FUNCTION_BLOCK PUBLIC FB_CylinderDriver EXTENDS FB_ComponentBase IMPLEMENTS ITF_Cylinder, ITFComponent
VAR_INPUT
	bSafetyOk				: BOOL; // Freigabe von Sicherheit
	
	bEnableHp				: BOOL;	// Freigabe Grundposition
	bEnableWp				: BOOL;	// Freigabe Arbeitsposition
END_VAR
VAR_OUTPUT
	// Zylinder ist in Grundstellung (verzögert)
	bIsInHp	: BOOL;
	// Zylinder ist in Arbeitsstellung (verzögert)
	bIsInWp	: BOOL;
	// Zylinder Ist-Position
	eActPos	: E_CylinderPosition;
END_VAR
VAR
	/// IO reference
	stIn 	: REFERENCE TO ST_CylinderDriverIn;
	stOut 	: REFERENCE TO ST_CylinderDriverOut;
	
	bWpSensor				: BOOL := TRUE;
	bHpSensor				: BOOL := TRUE;
	
	// private var's
	eReqPos					: E_CylinderPosition;	// Zylinder Soll-Position
	fPositionValidationTime	: TIME := T#300MS; 		// Verweilzeit bis die jeweilige Endlage bestätigt wird.
	tImpulseTime 			: TIME := T#0S; 		// Ansteuerzeit für Impulsventile (0 deaktiviert die Impulssteuerung)
	fSupervisionTime		: TIME := T#5S; 		// Verweilzeit nach Ventilansteuerung, bis die Zylinderendlage geprüft wird (0 deaktiviert die Überwachung)
	tonValveChange			: TON;					// Zeit seit Veränderung der Ventilstellung
	tonIsInHp				: TON;					// Verzögerung in Grundstellung
	tonIsInWp				: TON;					// Verzögerung in Arbeitsstellung
END_VAR

///
/// Cylinder driver FB
/// TP/www.rmth.at/06.2015
///

PROPERTY PUBLIC ActualPosition : E_CylinderPosition
GET
ActualPosition := eActPos;
END_GET
END_PROPERTY

PROPERTY PUBLIC EnableHp : BOOL
GET
EnableHp := bEnableHp;
END_GET
SET
bEnableHp := EnableHp;
END_SET
END_PROPERTY

PROPERTY PUBLIC EnableHpSensor : BOOL
GET
EnableHpSensor := bHpSensor;
END_GET
SET
bHpSensor := EnableHpSensor;
END_SET
END_PROPERTY

PROPERTY PUBLIC EnableWp : BOOL
GET
EnableWp := bEnableWp;
END_GET
SET
bEnableWp := EnableWp;
END_SET
END_PROPERTY

PROPERTY PUBLIC EnableWpSensor : BOOL
GET
EnableWpSensor := bWpSensor;
END_GET
SET
bWpSensor := EnableWpSensor;
END_SET
END_PROPERTY

METHOD FB_init : BOOL
VAR_INPUT
	bInitRetains : BOOL; // if TRUE, the retain variables are initialized (warm start / cold start)
	bInCopyCode : BOOL;  // if TRUE, the instance afterwards gets moved into the copy code (online change)
END_VAR
eTyp := E_ComponentType.eComponentType_Cylinder;
END_METHOD

// Ansteuerzeit für Impulsventile (0 deaktiviert die Impulssteuerung)
PROPERTY PUBLIC ImpulseTime : TIME
GET
// Ansteuerzeit für Impulsventile (0 deaktiviert die Impulssteuerung)
ImpulseTime := tImpulseTime;
END_GET
SET
// Ansteuerzeit für Impulsventile (0 deaktiviert die Impulssteuerung)
tImpulseTime := ImpulseTime;
END_SET
END_PROPERTY

/// Verweilzeit bis die jeweilige Endlage bestätigt wird.
PROPERTY PUBLIC PositionValidationTime : TIME
GET
/// Verweilzeit bis die jeweilige Endlage bestätigt wird.
PositionValidationTime := fPositionValidationTime;
END_GET
SET
/// Verweilzeit bis die jeweilige Endlage bestätigt wird.
fPositionValidationTime := PositionValidationTime;
END_SET
END_PROPERTY

PROPERTY PUBLIC RequestPosition : E_CylinderPosition
GET
RequestPosition := eReqPos;
END_GET
END_PROPERTY

METHOD Reset
VAR_INPUT
END_VAR
// base logic run
SUPER^.Reset();

//ToHP();
tonValveChange(IN := FALSE);
tonIsInHp(IN := FALSE);
tonIsInWp(IN := FALSE);

eState := E_ComponentState.eComponentState_ready;
END_METHOD

METHOD PUBLIC ResetValves
VAR_INPUT
END_VAR
IF NOT __ISVALIDREF(stOut) THEN
	sLastError := 'IO reference not set';
	eState := E_ComponentState.eComponentState_error;
	RETURN;
END_IF

// chk
IF NOT bSafetyOk THEN
	sClearText := 'Warte auf Sicherheit Ok';
	RETURN;
END_IF

eReqPos := eCylinderPosition_unknown;
stOut.bValveCylinderHp := FALSE;
stOut.bValveCylinderWp := FALSE;
tonValveChange(IN := FALSE);
END_METHOD

/// Run component logic
{attribute 'object_name' := 'Run'}
METHOD Run : E_ComponentState
// base logic run
Run := SUPER^.Run();

// chk
IF NOT (__ISVALIDREF(stIn) AND __ISVALIDREF(stOut)) THEN
	sLastError := 'IO reference not set';
	eState := E_ComponentState.eComponentState_error;
	RETURN;
END_IF



// definiere aktuelle Zylinderposition
IF (stIn.bCylinderSensorHp OR (NOT bHpSensor AND stOut.bValveCylinderHp)) AND NOT stIn.bCylinderSensorWp THEN
	eActPos := eCylinderPosition_hp;
ELSIF NOT stIn.bCylinderSensorHp AND (stIn.bCylinderSensorWp OR (NOT bWpSensor AND stOut.bValveCylinderWp)) THEN
	eActPos := eCylinderPosition_wp;
ELSE
	eActPos := eCylinderPosition_unknown;
END_IF

tonIsInHp(IN := (eActPos = eCylinderPosition_hp), PT := fPositionValidationTime);
bIsInHp := tonIsInHp.Q;

tonIsInWp(IN := (eActPos = eCylinderPosition_wp), PT := fPositionValidationTime);
bIsInWp := tonIsInWp.Q;

// Zeitmessung seit Veränderung der Ventilstellung 
tonValveChange(IN := TRUE, PT := tMaxTime);

// für Impulsventile (T#0S od. Wartungsmodus -> Funktion deaktiv)
IF tImpulseTime > T#0S AND tonValveChange.ET > tImpulseTime THEN
	stOut.bValveCylinderHp := FALSE;
	stOut.bValveCylinderWp := FALSE;
END_IF

// Zylinderüberwachung (T#0S -> Funktion deaktiv)
IF fSupervisionTime > T#0S AND tonValveChange.ET > fSupervisionTime AND eActPos <> eReqPos THEN
	IF eReqPos = eCylinderPosition_hp THEN
		sLastError := Concat(sName, ' Grundstellung nicht erreicht.');
		IF stIn.bCylinderSensorWp THEN
			sLastError := Concat(sLastError, ' Signal Arbeitsstellung steht noch an.');
		END_IF
		IF NOT stIn.bCylinderSensorHp THEN
			sLastError := Concat(sLastError, ' Signal Sensor Grundstellung fehlt.');
		END_IF
		IF __ISVALIDREF(fbEventLog) THEN		
			WriteError(E_Event.eEvent_none , sLastError);	
		END_IF
		eState := E_ComponentState.eComponentState_error;
	ELSIF eReqPos = eCylinderPosition_wp THEN
		sLastError := Concat(sName, ' Arbeitsstellung nicht erreicht.');
		IF stIn.bCylinderSensorHp THEN
			sLastError := Concat(sLastError, ' Signal Grundstellung steht noch an.');
		END_IF
		IF NOT stIn.bCylinderSensorWp THEN
			sLastError := Concat(sLastError, ' Signal Arbeitsstellung fehlt.');
		END_IF
		IF __ISVALIDREF(fbEventLog) THEN
			WriteError(E_Event.eEvent_none , sLastError);
		END_IF
		eState := E_ComponentState.eComponentState_error;
	END_IF
END_IF

//
END_METHOD

PROPERTY PUBLIC SafetyOk : BOOL
GET
SafetyOk := bSafetyOk;
END_GET
SET
bSafetyOk := SafetyOk;
END_SET
END_PROPERTY

PROPERTY PUBLIC SensorHp : BOOL
GET
IF __ISVALIDREF(stIn) THEN
	SensorHp := stIn.bCylinderSensorHp;
END_IF
END_GET
END_PROPERTY

PROPERTY PUBLIC SensorWp : BOOL
GET
IF __ISVALIDREF(stIn) THEN
	SensorWp := stIn.bCylinderSensorWp;
END_IF
END_GET
END_PROPERTY

METHOD PUBLIC SetImpulseTime
VAR_INPUT
	/// Ansteuerzeit für Impulsventile (0 deaktiviert die Impulssteuerung)
	tTime : TIME;
END_VAR
END_METHOD

/// Set up reference dependencies.
{attribute 'object_name' := 'SetIoReference'}
METHOD SetIoReference
VAR_IN_OUT
	stRefIn		: ST_CylinderDriverIn;
	stRefOut	: ST_CylinderDriverOut;
END_VAR
stIn 	REF= stRefIn;
stOut 	REF= stRefOut;
END_METHOD

/// Verweilzeit nach Ventilansteuerung, bis die Zylinderendlage geprüft wird (0 deaktiviert die Überwachung)
PROPERTY PUBLIC SupervisionTime : TIME
GET
/// Verweilzeit nach Ventilansteuerung, bis die Zylinderendlage geprüft wird (0 deaktiviert die Überwachung)
SupervisionTime := fSupervisionTime;
END_GET
SET
/// Verweilzeit nach Ventilansteuerung, bis die Zylinderendlage geprüft wird (0 deaktiviert die Überwachung)
fSupervisionTime := SupervisionTime;
END_SET
END_PROPERTY

METHOD PUBLIC ToHP
VAR_INPUT
END_VAR
IF NOT __ISVALIDREF(stOut) THEN
	sLastError := 'IO reference not set';
	eState := E_ComponentState.eComponentState_error;
	RETURN;
END_IF

// chk
IF NOT bSafetyOk THEN
	sClearText := 'Warte auf Sicherheit Ok';
	RETURN;
ELSIF NOT bEnableHp THEN
	sClearText := 'Warte auf Freigabe Hp';
	RETURN;
END_IF

eReqPos := eCylinderPosition_hp;
stOut.bValveCylinderHp := TRUE;
stOut.bValveCylinderWp := FALSE;
tonValveChange(IN := FALSE);
END_METHOD

METHOD PUBLIC ToWP
VAR_INPUT
END_VAR
IF NOT __ISVALIDREF(stOut) THEN
	sLastError := 'IO reference not set';
	eState := E_ComponentState.eComponentState_error;
	RETURN;
END_IF

// chk
IF NOT bSafetyOk THEN
	sClearText := 'Warte auf Sicherheit Ok';
	RETURN;
ELSIF NOT bEnableWp THEN
	sClearText := 'Warte auf Freigabe WP';
	RETURN;
END_IF

eReqPos := eCylinderPosition_wp;
stOut.bValveCylinderHp := FALSE;
stOut.bValveCylinderWp := TRUE;
tonValveChange(IN := FALSE);
END_METHOD

END_FUNCTION_BLOCK

(* stored: Version 1.1.0.1, ProductVersion 3.1.4022.9
   POU FB_CylinderDriver: Id {a82aae65-7938-479c-b543-36a2ecf1026e}, SpecialFunc None
   Folder Factory: Id {346f54fe-1c67-416c-8f69-6c95d1377e0a}
   Folder Properties: Id {280af190-36c4-4431-b31d-d2cb866e5894}
   Property ActualPosition: Id {044de178-debb-4265-b0ad-9e61c441a597}
   Get Get: Id {db805540-5ebb-454b-828f-16c80d784fc7}
   Property EnableHp: Id {6cf16ccf-9211-49e8-bdb2-da85e2b751b8}
   Get Get: Id {78c54a39-512b-45fc-a57d-9b8eddb92d98}
   Set Set: Id {603fafc5-ff53-478e-8d7d-d4ce84fc79b6}
   Property EnableHpSensor: Id {5e3a3ed7-0e74-47b4-8590-6a37261b3b12}
   Get Get: Id {c5015790-881a-491e-b71e-11d9f8f31897}
   Set Set: Id {09d89112-ffd7-44c3-9e9b-f65d1a7935cf}
   Property EnableWp: Id {24f24d54-7f29-4d1a-a366-81fcc2765573}
   Get Get: Id {948c9f3d-43bc-4ab7-b73b-bec0b9ce507f}
   Set Set: Id {a3bb4ec2-b5fb-4c42-b1c5-015f32a1fe44}
   Property EnableWpSensor: Id {f6fb1351-4d30-4807-a918-43d7f2fc822b}
   Get Get: Id {504bb3c9-b5b1-46a4-946b-207a2b0ad751}
   Set Set: Id {f814de94-6dbb-4e87-8e05-28a65841eab7}
   Method FB_init: Id {126f9f7c-a89d-46b1-8119-30f3ff4fb321}
   Property ImpulseTime: Id {2eb02d44-cb99-4d9d-9681-b66c53100d09}
   Get Get: Id {6ed0c4e4-6399-43ae-9774-f29f04703758}
   Set Set: Id {e9397767-16aa-4085-b446-123a1618e864}
   Property PositionValidationTime: Id {7f08aeaf-2435-46d4-b450-f973addc6b32}
   Get Get: Id {88b6b5e8-1110-404a-80dc-0b171fbc3189}
   Set Set: Id {be136f34-3f1e-478f-98f0-20843a0d200d}
   Property RequestPosition: Id {71c26901-5e60-43f8-8b28-291d5f1bbdef}
   Get Get: Id {6c63a25f-2cb8-40d6-b546-1dec372b987c}
   Method Reset: Id {9554fe57-0fe8-45d4-8baf-0ce375ce1131}
   Method ResetValves: Id {935e2cf7-22ae-418b-9435-aa75101323e7}
   Method Run: Id {cc7b2bfb-3730-4f25-913f-7c5dc50032db}
   Property SafetyOk: Id {0d868bd4-59ca-491f-a4ed-46ca277f2418}
   Get Get: Id {e3fa39fa-e134-4c18-adc3-e379a21e3d69}
   Set Set: Id {14d9cd63-7d2f-4b36-8775-fcf415ae1012}
   Property SensorHp: Id {2980b765-9a95-4a0c-87d3-a92f58655219}
   Get Get: Id {eb8e15c7-1790-4971-9e70-646c8af40911}
   Property SensorWp: Id {c88d5ca0-4b38-448d-a9d5-a27dc5a9f0ac}
   Get Get: Id {97a1cec2-6595-4679-a436-f81ccd6fa7eb}
   Method SetImpulseTime: Id {421100bf-2256-4d9c-98fb-a2fdf3d51a44}
   Method SetIoReference: Id {20cf7886-d27d-4c9d-a118-821f51be2f18}
   Property SupervisionTime: Id {943f890e-c86e-4134-a850-43379d5cf33a}
   Get Get: Id {81dc8b15-6348-4cf1-9d43-542913353ca2}
   Set Set: Id {e051b8ba-2f3f-4166-bc1c-40deb4bbf6a7}
   Method ToHP: Id {97e530d7-0b7a-4d4c-8a20-ce952bab4715}
   Method ToWP: Id {7b3857aa-191a-43c9-bb8a-f0eb6e378844} *)
